FUNCTION_BLOCK ADD (* Add *)
  (* Standard: 61499-2 *)
  (* Version 1.0, 02.01.2011, gsha041, UoA, Initial Version *)
  (* Compiler header: package fb.rt.UoA; *)
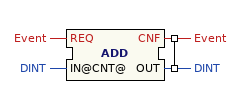
  EVENT_INPUT
    REQ; (* Normal Execution Request *)
  END_EVENT
  EVENT_OUTPUT
    CNF WITH OUT; (* Execution Confirmation *)
  END_EVENT
  VAR_INPUT
    IN@CNT@ : DINT; (* Argument *)
  END_VAR
  VAR_OUTPUT
    OUT : DINT; (* Result: IN1 + IN2 + ... *)
  END_VAR
END_FUNCTION_BLOCK
